// TIA Portal V20 export
ORGANIZATION_BLOCK "CyclicInterruptReceiveData"   // OB30, LAD, CyclicInterrupt
TITLE = Cyclic data trasfer to partner PLC
// Template v0.1
// stored: Namespace Safety, SetENOAutomatically false
   VAR_INPUT
      Initial_Call : Bool;   // Initial call of this OB
      Event_Count : Int;   // Events discarded
   END_VAR
   VAR_TEMP
      statErrorRcvAck : Word;
      statErrorRcvData : Word;
   END_VAR
BEGIN

REGION Network 1: Transfer F-data and ackowledge signal to BA10AC1
   // V1.0  25.05.04  test program
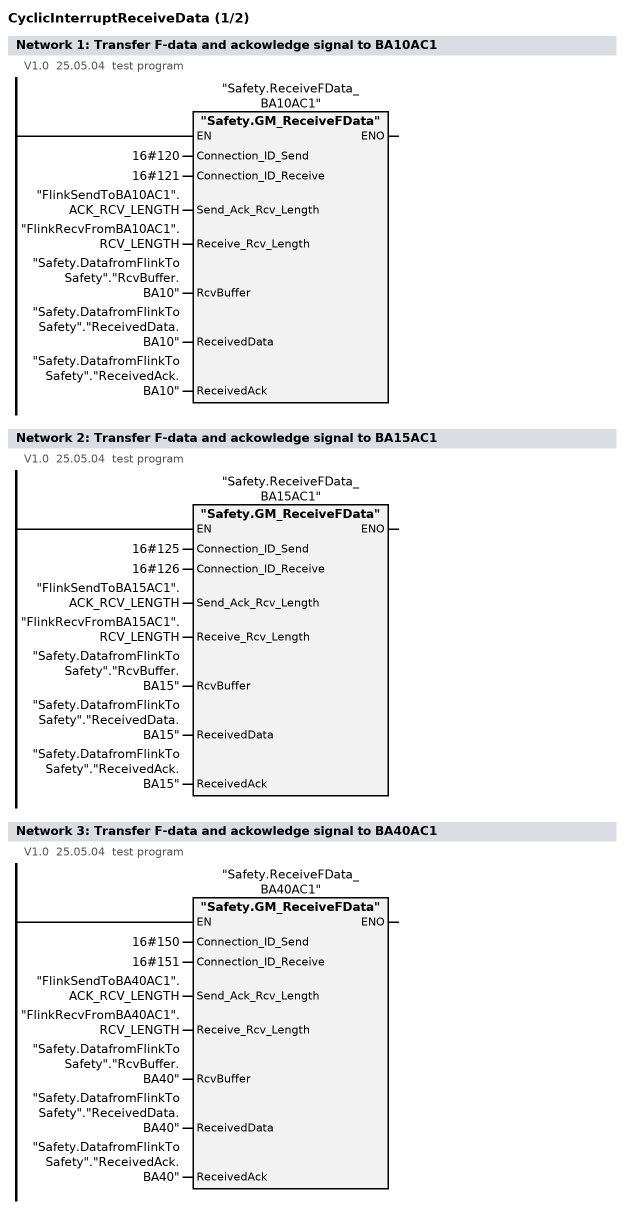
   RUNG wire#powerrail
      "Safety.ReceiveFData_BA10AC1"(Connection_ID_Send := 16#120, Connection_ID_Receive := 16#121, Send_Ack_Rcv_Length := "FlinkSendToBA10AC1".ACK_RCV_LENGTH, Receive_Rcv_Length := "FlinkRecvFromBA10AC1".RCV_LENGTH, RcvBuffer := "Safety.DatafromFlinkToSafety"."RcvBuffer.BA10", ReceivedData := "Safety.DatafromFlinkToSafety"."ReceivedData.BA10", ReceivedAck := "Safety.DatafromFlinkToSafety"."ReceivedAck.BA10")
   END_RUNG
   // the same network as SCL:
   "Safety.ReceiveFData_BA10AC1"(Connection_ID_Send := 16#120,   // "Safety.GM_ReceiveFData"
                           Connection_ID_Receive := 16#121,
                           Send_Ack_Rcv_Length := "FlinkSendToBA10AC1".ACK_RCV_LENGTH,
                           Receive_Rcv_Length := "FlinkRecvFromBA10AC1".RCV_LENGTH,
                           RcvBuffer := "Safety.DatafromFlinkToSafety"."RcvBuffer.BA10",
                           ReceivedData := "Safety.DatafromFlinkToSafety"."ReceivedData.BA10",
                           ReceivedAck := "Safety.DatafromFlinkToSafety"."ReceivedAck.BA10");
END_REGION

REGION Network 2: Transfer F-data and ackowledge signal to BA15AC1
   // V1.0  25.05.04  test program
   RUNG wire#powerrail
      "Safety.ReceiveFData_BA15AC1"(Connection_ID_Send := 16#125, Connection_ID_Receive := 16#126, Send_Ack_Rcv_Length := "FlinkSendToBA15AC1".ACK_RCV_LENGTH, Receive_Rcv_Length := "FlinkRecvFromBA15AC1".RCV_LENGTH, RcvBuffer := "Safety.DatafromFlinkToSafety"."RcvBuffer.BA15", ReceivedData := "Safety.DatafromFlinkToSafety"."ReceivedData.BA15", ReceivedAck := "Safety.DatafromFlinkToSafety"."ReceivedAck.BA15")
   END_RUNG
   // the same network as SCL:
   "Safety.ReceiveFData_BA15AC1"(Connection_ID_Send := 16#125,   // "Safety.GM_ReceiveFData"
                           Connection_ID_Receive := 16#126,
                           Send_Ack_Rcv_Length := "FlinkSendToBA15AC1".ACK_RCV_LENGTH,
                           Receive_Rcv_Length := "FlinkRecvFromBA15AC1".RCV_LENGTH,
                           RcvBuffer := "Safety.DatafromFlinkToSafety"."RcvBuffer.BA15",
                           ReceivedData := "Safety.DatafromFlinkToSafety"."ReceivedData.BA15",
                           ReceivedAck := "Safety.DatafromFlinkToSafety"."ReceivedAck.BA15");
END_REGION

REGION Network 3: Transfer F-data and ackowledge signal to BA40AC1
   // V1.0  25.05.04  test program
   RUNG wire#powerrail
      "Safety.ReceiveFData_BA40AC1"(Connection_ID_Send := 16#150, Connection_ID_Receive := 16#151, Send_Ack_Rcv_Length := "FlinkSendToBA40AC1".ACK_RCV_LENGTH, Receive_Rcv_Length := "FlinkRecvFromBA40AC1".RCV_LENGTH, RcvBuffer := "Safety.DatafromFlinkToSafety"."RcvBuffer.BA40", ReceivedData := "Safety.DatafromFlinkToSafety"."ReceivedData.BA40", ReceivedAck := "Safety.DatafromFlinkToSafety"."ReceivedAck.BA40")
   END_RUNG
   // the same network as SCL:
   "Safety.ReceiveFData_BA40AC1"(Connection_ID_Send := 16#150,   // "Safety.GM_ReceiveFData"
                           Connection_ID_Receive := 16#151,
                           Send_Ack_Rcv_Length := "FlinkSendToBA40AC1".ACK_RCV_LENGTH,
                           Receive_Rcv_Length := "FlinkRecvFromBA40AC1".RCV_LENGTH,
                           RcvBuffer := "Safety.DatafromFlinkToSafety"."RcvBuffer.BA40",
                           ReceivedData := "Safety.DatafromFlinkToSafety"."ReceivedData.BA40",
                           ReceivedAck := "Safety.DatafromFlinkToSafety"."ReceivedAck.BA40");
END_REGION

REGION Network 4: Transfer F-data and ackowledge signal to BA60AC1
   // V1.0  25.05.04  test program
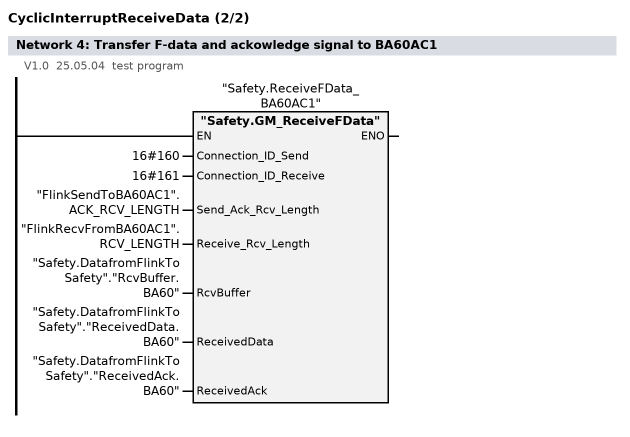
   RUNG wire#powerrail
      "Safety.ReceiveFData_BA60AC1"(Connection_ID_Send := 16#160, Connection_ID_Receive := 16#161, Send_Ack_Rcv_Length := "FlinkSendToBA60AC1".ACK_RCV_LENGTH, Receive_Rcv_Length := "FlinkRecvFromBA60AC1".RCV_LENGTH, RcvBuffer := "Safety.DatafromFlinkToSafety"."RcvBuffer.BA60", ReceivedData := "Safety.DatafromFlinkToSafety"."ReceivedData.BA60", ReceivedAck := "Safety.DatafromFlinkToSafety"."ReceivedAck.BA60")
   END_RUNG
   // the same network as SCL:
   "Safety.ReceiveFData_BA60AC1"(Connection_ID_Send := 16#160,   // "Safety.GM_ReceiveFData"
                           Connection_ID_Receive := 16#161,
                           Send_Ack_Rcv_Length := "FlinkSendToBA60AC1".ACK_RCV_LENGTH,
                           Receive_Rcv_Length := "FlinkRecvFromBA60AC1".RCV_LENGTH,
                           RcvBuffer := "Safety.DatafromFlinkToSafety"."RcvBuffer.BA60",
                           ReceivedData := "Safety.DatafromFlinkToSafety"."ReceivedData.BA60",
                           ReceivedAck := "Safety.DatafromFlinkToSafety"."ReceivedAck.BA60");
END_REGION
END_ORGANIZATION_BLOCK
